PROGRAM MAIN
VAR
END_VAR

END_PROGRAM

(* stored: Version 1.1.0.1
   POU MAIN: Id {302ddb90-5f4b-40d7-a128-f024b91f60a8} *)
